FUNCTION_BLOCK FB_TestHTTP_Mindsphere_AcquireAAT
VAR_INPUT
	bSend				: BOOL;
END_VAR
VAR_IN_OUT
	fbClient			: FB_IotHttpClient;
END_VAR
VAR_OUTPUT
	bBusy				: BOOL;
	bError				: BOOL;
END_VAR
VAR	
	fbRequest			: FB_IotHttpRequest;
	fbHeader			: FB_IotHttpHeaderFieldMap;
	fbJson				: FB_JsonDomParser;
	nState				: UDINT;
	RisingEdge			: R_TRIG;
	
	bGetContentResult	: BOOL;
	sContent			: STRING(2048);
	
	bGetJsonResult		: BOOL;
	jsonDoc				: SJsonValue;
	jsonVal				: SJsonValue;
	sResultValue		: STRING;
	
	nReqCount			: UDINT;
	nResCount			: UDINT;
	nValidResCount		: UDINT;
	nErrCount			: UDINT;	
END_VAR

RisingEdge(CLK:= bSend);
CASE nState OF
0:		
	IF RisingEdge.Q THEN
		sContent := 'grant_type=client_credentials&client_assertion_type=urn:ietf:params:oauth:client-assertion-type:jwt-bearer&client_assertion=eyJ0eXAiOiJKV1QiLCJhbGciOiJIUzI1NiJ9.eyJpc3MiOiI5NTZjY2UzNjA1YjE0MjA4OTAwOTVlNTBlMmIxMWUxNyIsInN1YiI6Ijk1NmNjZTM2MDViMTQyMDg5MDA5NWU1MGUyYjExZTE3IiwiYXVkIjpbInNvdXRoZ2F0ZSJdLCJpYXQiOjE1ODIxOTI2NjEsIm5iZiI6MTU4MjE5MjY2MSwiZXhwIjoxNTgyMTkzNjYxLCJqdGkiOiJjNDJlYjNiYy04NjI2LTQ3ZDktOTRjYy01MWE0OGQ3ZTc3YjMiLCJ0ZW4iOiJiZWNraG9mZiIsInNjaGVtYXMiOlsidXJuOnNpZW1lbnM6bWluZHNwaGVyZTp2MSJdfQ.LZcYDd38oRX1rdwGeBuqJVy5S4ja4Bmo5lvTW-EloP4';
		fbHeader.AddField('Content-Type', 'application/x-www-form-urlencoded', FALSE);
		IF fbRequest.SendRequest(sUri:= '/api/agentmanagement/v3/oauth/token', fbClient:= fbClient, eRequestType:= ETcIotHttpRequestType.HTTP_POST, pContent:= ADR(sContent), nContentSize:= LEN2(ADR(sContent)), fbHeader:= fbHeader) THEN				
			nState:= 1;
			nReqCount:= nReqCount+1;
			bBusy:= TRUE;
			bError:= FALSE;
		END_IF					
	END_IF
1:
	IF NOT fbRequest.bBusy THEN
		bError:= TRUE;
		IF NOT fbRequest.bError THEN				 				
			bGetContentResult:= fbRequest.GetContent(pContent:= ADR(sContent), nContentSize:= SIZEOF(sContent), bSetNullTermination:= TRUE);	
			IF fbRequest.nStatusCode >= 200 AND fbRequest.nStatusCode < 300 THEN
				bGetJsonResult:= FALSE;
				jsonDoc:= fbRequest.GetJsonDomContent(fbJson);				
				(* Parse AAT API Call response in order to acquire:
					access_token
					token_type
					expires_in
					scope
					jti 
				*)
				nResCount:= nResCount+1;					
			END_IF				
		END_IF
		nState:= 0;
		bBusy:= FALSE;
		IF bError THEN
			nErrCount:= nErrCount+1;
		END_IF		
	END_IF  	
END_CASE

END_FUNCTION_BLOCK

(* stored: Version 1.1.0.1, ProductVersion 3.1.4024.3
   POU FB_TestHTTP_Mindsphere_AcquireAAT: Id {d04a8356-6530-46c2-a2e9-d1ad96709113}, SpecialFunc None *)
